(* IEC 61131-3 sources: stGeo/src/Functions, 4 files *)

(* ---- CirclesInTriangle.st ---- *)
TYPE CirclesInTriangleError :
    (
        NO_ERROR,
        ROWS_EXCEEDED
    );
END_TYPE

FUNCTION CirclesInTriangle : CirclesInTriangleError
    VAR_INPUT
        Radius : LREAL := 1.0;
        Rows : UINT := 5;
        // possibly set max rows and
    END_VAR
    VAR_OUTPUT
       Points : ARRAY [0..65] OF XYPoint;
    END_VAR
    VAR
        RowLength : UINT := 0;
        RowOffset : XYPoint;
        Remaining : UINT;
        I : UINT;
        T60Rad : LREAL;
        PointsIndex : UINT := 0;
        XGap : LREAL;
    END_VAR
    VAR
        CONSTANT MAX_ROWS : UINT := 11;
    END_VAR

    IF Rows > MAX_ROWS THEN
       CirclesInTriangle := CirclesInTriangleError#ROWS_EXCEEDED;
       RETURN;
    END_IF
        T60Rad := TAN(RAD(60)) * Radius;
        XGap := LREAL#2.0 * Radius;
    FOR I := 0 TO Rows -1 DO
        RowLength := RowLength + 1;
        Remaining := RowLength;
        WHILE Remaining > 0 DO
            Points[PointsIndex].X := RowOffset.X + (RowLength - Remaining ) * XGap;
            Points[PointsIndex].Y := RowOffset.Y;
            Remaining := Remaining - 1;
            PointsIndex := PointsIndex + 1;
        END_WHILE
        RowOffset.Y := RowOffset.Y + T60Rad;
        RowOffset.X := RowOffset.X - Radius;
    END_FOR
    CirclesInTriangle := CirclesInTriangleError#NO_ERROR;
END_FUNCTION

(* ---- RotateSquarePoints.st ---- *)
FUNCTION RotateSquarePoints : XYPoints
VAR_IN_OUT
    Square : XYPoints;
END_VAR
VAR
   X : LREAL;
   Y : LREAL;
   I : INT;
END_VAR
FOR I := 0 TO 3 DO
    X := Square[I].X;
    Y := Square[I].Y;
    Square[I] := RotateXY(
    X := X,
    Y := Y,
    THETA := 90.0
    );
END_FOR
RotateSquarePoints := Square;
END_FUNCTION

(* ---- RotateXY.st ---- *)
FUNCTION RotateXY : XYPoint
VAR_INPUT
    X : LREAL;
    Y : LREAL;
    THETA : LREAL;
END_VAR
VAR
    Out : XYPoint;
    SinM : LREAL;
    CosM : LREAL;
    THETA_RAD : LREAL;
END_VAR

   THETA_RAD := REAL_TO_LREAL(
    RAD(
        LREAL_TO_REAL(THETA)
        )
    );
   SinM := SIN(THETA_RAD);
   Cosm := COS(THETA_RAD);
   Out.X := X * CosM - Y * SinM;
   Out.Y := X * SinM + Y * CosM;
   RotateXY := Out;
END_FUNCTION

(* ---- SquarePoints.st ---- *)
FUNCTION SquarePoints : XYPoints
VAR_OUTPUT
    //Square : Array[0..1] of LREAL;//XYPoints;
END_VAR
VAR_INPUT
    Length : LREAL := 5.0;

END_VAR
VAR
   Zero : LREAL := 0.0;
   Square : XYPoints;
END_VAR

    Square[0].X := Zero;
    Square[0].Y := Length;
    Square[1].X := Length;
    Square[1].Y := Length;
    Square[2].X := Length;
    Square[2].Y := Zero;
    Square[3].X := Zero;
    Square[3].Y := Zero;
    SquarePoints := Square;
END_FUNCTION
